FUNCTION_BLOCK FlushSludgeBuffer (* CAT Function Block Type *)
  (* Standard: 61499-2 *)
  (* Version 0.0, 6/19/2026, Schneider Electric, template *)
  PACKAGE SE.Nereda;
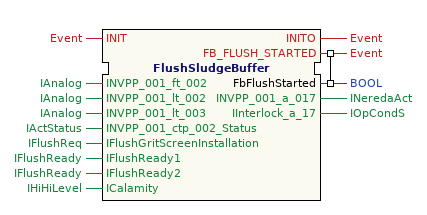
  EVENT_INPUT
    INIT;
  END_EVENT
  EVENT_OUTPUT
    INITO;
    FB_FLUSH_STARTED WITH FbFlushStarted;
  END_EVENT
  VAR_OUTPUT
    FbFlushStarted : BOOL;
  END_VAR
  SOCKETS
    INVPP_001_ft_002 : IAnalog;
    INVPP_001_lt_002 : IAnalog;
    INVPP_001_lt_003 : IAnalog;
    INVPP_001_ctp_002_Status : IActStatus;
    IFlushGritScreenInstallation : IFlushReq;
    IFlushReady1 : IFlushReady;
    IFlushReady2 : IFlushReady;
    ICalamity : IHiHiLevel;
  END_SOCKETS
  PLUGS
    INVPP_001_a_017 : INeredaAct;
  END_PLUGS
  PLUGS
    IInterlock_a_17 : IOpCondS; (* Condition summary chain output to downstream block *)
  END_PLUGS
  (* 01 - FUNCTIONNAL INPUT INTERFACE *)
  (* 00 - INITIALIZATION *)
  (* 05 - LOGIC *)
  (* 06 - HMI INTERFACE *)
  (* 03 - FIELD INTERFACE *)
  (* Grit Screens Flush Conditions *)
  (* 02 - FUNCTIONNAL OUTPUT INTERFACE *)
  (* Grit Screens Flush Control *)
  (* Interlock *)
  FBS
    FlushConditions : FlushCdt(pin_AD4F1D04748929A2 := 'Effluent Level is ok', pin_D80C7C0ABBECCDAB := 'Sludge Buffer Flushing', pin_E55C299A5BCFE2A5 := 'NVPP 001 a-- 017 is Available', pin_4F5AA965534A9167 := 'No Low Low Flow Alarm (Effluent Pump)', pin_D8438E8592CCBB68 := 'Effluent Pump is Ready', pin_F9CA602A9987631B := 'Flushing Parametrization is Done', pin_D946781DFBE190E0 := 'No Hi Level - Sludge Buffer', pin_2F47EB70426E0A5E := 'Flush Level Sp reached', pin_2D24E9AB41BE5BDB := TRUE, pin_EDFD852BF7F500FC := '');
    IThis : FlushSludgeBuffer_HMI(QI := TRUE);
    NVPP_001_lt_002_Status : decodeStatus; {SET_ATTRIBUTE(Configuration.Component.HideUnusedPorts, )}
    NotLowLevel : NOT_42C76073DCEB1A7A; {SET_ATTRIBUTE(Configuration.GenericFBType.InterfaceParams, Runtime.Standard#CNT:=1;OUT${CNT$}:BOOL)}
    GritScreensFlushControl : FlushingManagerSLB;
    Valve016_002Cmd : boolValueChanged;
    DurationSp : COMPARE_231D1C451B8C01CD0(IN2 := T#0ms); {SET_ATTRIBUTE(Configuration.GenericFBType.InterfaceParams, Runtime.Standard#CNT:=2;IN${CNT$}:TIME)} {SET_ATTRIBUTE(Configuration.Component.HideUnusedPorts, )}
    ConfigDone : AND_88A3DD8EC65DD11C; {SET_ATTRIBUTE(Configuration.GenericFBType.InterfaceParams, Runtime.Standard#CNT:=2;OUT:BOOL)}
    NVPP_001_ft_002_Status : decodeStatus; {SET_ATTRIBUTE(Configuration.Component.HideUnusedPorts, )}
    NotLowLowFlow : NOT_42C76073DCEB1A7A; {SET_ATTRIBUTE(Configuration.GenericFBType.InterfaceParams, Runtime.Standard#CNT:=1;OUT${CNT$}:BOOL)}
    CmdValve016_002 : BOOL2INT;
    FlowSp : COMPARE_1329C2AB45109BAAB(IN2 := 0); {SET_ATTRIBUTE(Configuration.GenericFBType.InterfaceParams, Runtime.Standard#CNT:=2;IN${CNT$}:REAL)} {SET_ATTRIBUTE(Configuration.Component.HideUnusedPorts, )}
    ForceStopSmooth : boolValueChanged;
    ForceStop : OR_NOT(pin_5391A9290C426EAD := FALSE, pin_0C6244A1FA53F771 := FALSE, pin_C718A4E0F6B1A5AF := FALSE, pin_F9B6B2F79CE46D8A := FALSE, pin_892061249439E371 := FALSE, pin_A17BF02B1ECA9592 := FALSE, pin_8BCAE36E149A36F2 := FALSE, pin_58FCE90E3A313BCD := TRUE, pin_7433DE8044744DCF := FALSE, pin_8555750E45CD1B5C := TRUE);
    ResetBtns : RESET_BTNs;
    NVPP_001_lt_003_Status : decodeStatus; {SET_ATTRIBUTE(Configuration.Component.HideUnusedPorts, )}
    NoHiLevel : NOT_42C76073DCEB1A7A; {SET_ATTRIBUTE(Configuration.GenericFBType.InterfaceParams, Runtime.Standard#CNT:=1;OUT${CNT$}:BOOL)}
    FlushStartLevelSp : COMPARE_1329C2AB45109BAAB; {SET_ATTRIBUTE(Configuration.GenericFBType.InterfaceParams, Runtime.Standard#CNT:=2;IN${CNT$}:REAL)}
    HighHighLevel_Calamity : ilckCondItem(CondCause := Active1);
    HighHighCalamity : OR_88A3DD8EC65DD11C; {SET_ATTRIBUTE(Configuration.GenericFBType.InterfaceParams, Runtime.Standard#CNT:=2;OUT:BOOL)}
    Wait : E_DELAY(DT := T#10s);
    GSsORGSsStarted : OR_88A3DD8EC65DD11C; {SET_ATTRIBUTE(Configuration.GenericFBType.InterfaceParams, Runtime.Standard#CNT:=2;OUT:BOOL)}
    DurationTime : E_DELAY_HOLD_V_D;
    Smooth : boolValueChanged;
    GSsORGSsFlushStarted : OR_88A3DD8EC65DD11C; {SET_ATTRIBUTE(Configuration.GenericFBType.InterfaceParams, Runtime.Standard#CNT:=2;OUT:BOOL)}
    Smooth1 : boolValueChanged;
  END_FBS
  EVENT_CONNECTIONS
    INVPP_001_lt_002.REQ_STATUS TO NVPP_001_lt_002_Status.REQ;
    NVPP_001_lt_002_Status.CNF TO NotLowLevel.REQ;
    NotLowLowFlow.CNF TO DurationSp.REQ;
    DurationSp.CNF TO FlowSp.REQ;
    INVPP_001_ft_002.REQ_STATUS TO NVPP_001_ft_002_Status.REQ;
    NVPP_001_ft_002_Status.CNF TO NotLowLevel.REQ;
    NotLowLevel.CNF TO NotLowLowFlow.REQ;
    FlushConditions.E74FDFC5C9E17061 TO INITO;
    DurationTime.INITO TO FlushConditions.7689825C23C7E3C1;
    INVPP_001_a_017.9CD053F8408797ED TO GritScreensFlushControl.17EF565317C21577;
    DurationTime.1457E63E0C241C83 TO GritScreensFlushControl.6BFDB43937C58B53;
    GritScreensFlushControl.FB17218C6899B6C2 TO FB_FLUSH_STARTED;
    GritScreensFlushControl.7C8478AB3E0AC40C TO Valve016_002Cmd.REQ;
    GritScreensFlushControl.4439D0346679ABD7 TO IFlushGritScreenInstallation.058C8BB5EF4C4954;
    GritScreensFlushControl.CNF_FLUSH_START TO DurationTime.START;
    GritScreensFlushControl.CNF_FLUSH_STOP TO DurationTime.STOP;
    Valve016_002Cmd.CHD TO CmdValve016_002.DD5870AA881150BB;
    CmdValve016_002.6FC99A5BD1C38561 TO INVPP_001_a_017.0F1CDF9A9B4A227A;
    INVPP_001_a_017.CC753684FA882790 TO NotLowLevel.REQ;
    FlushStartLevelSp.CNF TO FlushConditions.C4A26A2931936C6C;
    ForceStop.5E2BC6C1897CC372 TO ForceStopSmooth.REQ;
    FlushConditions.144BD964598CDC30 TO GritScreensFlushControl.D472A6751679CB56;
    INIT TO IThis.1EF99DCB15A49BE4;
    GritScreensFlushControl.GRAPH TO IThis.623B20E659F013A2;
    FlushConditions.E74FDFC5C9E17061 TO IThis.6CA585F7EA2251CC;
    ResetBtns.920962203CA54948 TO IThis.BC4D95AF9C39047B;
    IThis.97A2502A32C860AE TO DurationTime.INIT;
    IThis.40B0BCBFC46CBB6D TO NotLowLevel.REQ;
    IThis.40B0BCBFC46CBB6D TO IFlushGritScreenInstallation.A591EFC748C65FB0;
    IThis.40B0BCBFC46CBB6D TO DurationTime.8C325F07198FCB13;
    IThis.C0957A1C40CEA3B4 TO GritScreensFlushControl.F40A51463574875E;
    IThis.C0957A1C40CEA3B4 TO ResetBtns.AB695E9A35A20E19;
    GritScreensFlushControl.F622B0785D87399D TO IFlushGritScreenInstallation.91C62E5F9EC3AD97;
    INVPP_001_ctp_002_Status.14377629A1F197A9 TO NotLowLevel.REQ;
    IFlushGritScreenInstallation.158ACCEF11EA11F4 TO GritScreensFlushControl.2E9E428AF53DA484;
    INVPP_001_lt_003.REQ_STATUS TO NVPP_001_lt_003_Status.REQ;
    NVPP_001_lt_003_Status.CNF TO NotLowLevel.REQ;
    ForceStopSmooth.CNF TO NoHiLevel.REQ;
    NoHiLevel.CNF TO FlushStartLevelSp.REQ;
    INVPP_001_lt_003.REQ TO NotLowLevel.REQ;
    FlushStartLevelSp.CNF TO GritScreensFlushControl.7CCDF8BA66CD247C;
    HighHighCalamity.CNF TO HighHighLevel_Calamity.REQ;
    ICalamity.15126F43E529BB4F TO HighHighCalamity.REQ;
    FlowSp.CNF TO ConfigDone.REQ;
    ConfigDone.CNF TO ForceStop.AE1B4DCC5DF54611;
    GritScreensFlushControl.9781ED32849F99B4 TO Wait.START;
    Wait.EO TO GritScreensFlushControl.F24FFDC5DA37517C;
    IFlushReady1.EB400628E9D6A506 TO GSsORGSsStarted.REQ;
    IFlushReady2.EB400628E9D6A506 TO GSsORGSsStarted.REQ;
    GritScreensFlushControl.33239982CC8E7419 TO DurationTime.46FF7A1A69D9FEE0;
    GSsORGSsStarted.CNF TO Smooth.REQ;
    Smooth.CHD TO GritScreensFlushControl.D472A6751679CB56;
    IFlushReady1.A6EF038FCF65FFCE TO GSsORGSsFlushStarted.REQ;
    IFlushReady2.A6EF038FCF65FFCE TO GSsORGSsFlushStarted.REQ;
    GSsORGSsFlushStarted.CNF TO Smooth1.REQ;
    Smooth1.CHD TO GritScreensFlushControl.C7A0D51879FE2FD9;
  END_CONNECTIONS
  DATA_CONNECTIONS
    INVPP_001_lt_002.Status TO NVPP_001_lt_002_Status.Status;
    NVPP_001_lt_002_Status.LoAlarm TO NotLowLevel.IN1;
    INVPP_001_ft_002.Status TO NVPP_001_ft_002_Status.Status;
    NVPP_001_ft_002_Status.LoLoAlarm TO NotLowLowFlow.IN1;
    NotLowLevel.OUT1 TO FlushConditions.22A84A30EE8DD605;
    INVPP_001_a_017.8A8A07EFCDA1443C TO FlushConditions.4ED40FD24D2392DA;
    NotLowLowFlow.OUT1 TO FlushConditions.504E64E2CDCF5D86;
    INVPP_001_ctp_002_Status.9E0B44559326BEAF TO FlushConditions.9BB2492C130556E4;
    GritScreensFlushControl.7925856953128FBE TO FbFlushStarted;
    GritScreensFlushControl.6EFD4A5711C4475D TO Valve016_002Cmd.Input;
    GritScreensFlushControl.D35FF54DD8CD3DCD TO IFlushGritScreenInstallation.78ED129B4768A8A1;
    GritScreensFlushControl.809D6A4978DE08CF TO IFlushGritScreenInstallation.23612E77D592C190;
    Valve016_002Cmd.Output TO CmdValve016_002.4573FC8F228EB71D;
    DurationTime.716D3F3042596C89 TO GritScreensFlushControl.FlushDurationDone;
    INVPP_001_a_017.7F6CC7FEB9223DF3 TO GritScreensFlushControl.B4CCB3C919A81AAD;
    INVPP_001_a_017.A8D6C4A1FDCCA991 TO GritScreensFlushControl.927265D5AE017F25;
    IFlushGritScreenInstallation.309BBEDA7DF51DE0 TO GritScreensFlushControl.EB78D4EC51374885;
    IFlushGritScreenInstallation.E3447F193E0C5923 TO GritScreensFlushControl.8C9A5C84A4BBC11A;
    IFlushGritScreenInstallation.102FEFFE81A835E5 TO GritScreensFlushControl.BE830E3A77806910;
    IFlushGritScreenInstallation.32E78DF7D9CBD985 TO GritScreensFlushControl.CA6B1E62BFF3D73B;
    CmdValve016_002.A6DEF5F9C27C1848 TO INVPP_001_a_017.710D7FC54EE3F35A;
    ForceStop.39A6EB2EA34CB8B9 TO ForceStopSmooth.Input;
    NotLowLevel.OUT1 TO ForceStop.305F82B0106D312B;
    INVPP_001_a_017.8A8A07EFCDA1443C TO ForceStop.DD1680AE8DA8DF87;
    NotLowLowFlow.OUT1 TO ForceStop.92ECDEDDB24CC262;
    INVPP_001_ctp_002_Status.9E0B44559326BEAF TO ForceStop.2CF1E7F52666F162;
    FlushConditions.5C1922DA22925005 TO GritScreensFlushControl.EnableOperation;
    GritScreensFlushControl.Grafcet TO IThis.4EF02231C06E8D13;
    IThis.1AA6078AD289AF22 TO DurationSp.IN1;
    IThis.1AA6078AD289AF22 TO DurationTime.DT1;
    IThis.3E1384426DD858B0 TO FlowSp.IN1;
    IThis.3E1384426DD858B0 TO IFlushGritScreenInstallation.34B76CCA964D89EE;
    IThis.CEC3C53B3ACE8E6D TO GritScreensFlushControl.0FA765E9822F7BA9;
    IThis.CEC3C53B3ACE8E6D TO ResetBtns.479D4538AEFD6EE1;
    IThis.1BFB680DD0A7C843 TO GritScreensFlushControl.3C22F17908DBA162;
    GritScreensFlushControl.51D0A2C29DC62FA2 TO IFlushGritScreenInstallation.B5CD30493D22784A;
    GritScreensFlushControl.7AB11AE4573B259E TO IFlushGritScreenInstallation.10050E1891596878;
    IFlushGritScreenInstallation.0154EF4D281C90FC TO GritScreensFlushControl.9CD632B5AC2CF415;
    INVPP_001_lt_003.Status TO NVPP_001_lt_003_Status.Status;
    NVPP_001_lt_003_Status.HiAlarm TO NoHiLevel.IN1;
    NoHiLevel.OUT1 TO FlushConditions.4E3CFAB7818DC81F;
    FlushStartLevelSp.LE TO FlushConditions.47969CBC2D520AAD;
    INVPP_001_lt_003.Value TO FlushStartLevelSp.IN1;
    IThis.34A2F2095903B30B TO FlushStartLevelSp.IN2;
    FlushStartLevelSp.GT TO GritScreensFlushControl.336396CDA8290477;
    FlushStartLevelSp.LE TO GritScreensFlushControl.B610A3A56F10FBA2;
    HighHighCalamity.OUT TO HighHighLevel_Calamity.CondSignal;
    ICalamity.C818324478A2F205 TO HighHighCalamity.IN1;
    ICalamity.96B50ADF37756FFC TO HighHighCalamity.IN2;
    DurationSp.NE TO ConfigDone.IN1;
    FlowSp.NE TO ConfigDone.IN2;
    ConfigDone.OUT TO FlushConditions.9D55FD7AD1246DA2;
    ConfigDone.OUT TO ForceStop.4997B302A4472F6A;
    IFlushGritScreenInstallation.F75B2D6279DB7772 TO GritScreensFlushControl.AED40E274B455BA3;
    IFlushGritScreenInstallation.FBD19C5680BE3A13 TO GritScreensFlushControl.266B23EDF02E98D5;
    IFlushReady1.948E4422D799D3D4 TO GSsORGSsStarted.IN1;
    IFlushReady2.948E4422D799D3D4 TO GSsORGSsStarted.IN2;
    Smooth.Output TO GritScreensFlushControl.6757599E742CC6CD;
    GritScreensFlushControl.FDBF246FF450FFC3 TO DurationTime.5F12F87EEE9002AF;
    GSsORGSsStarted.OUT TO Smooth.Input;
    IFlushReady1.3B406C848FF944CA TO GSsORGSsFlushStarted.IN1;
    IFlushReady2.3B406C848FF944CA TO GSsORGSsFlushStarted.IN2;
    GSsORGSsFlushStarted.OUT TO Smooth1.Input;
    Smooth1.Output TO GritScreensFlushControl.1290DB47BB4481FA;
  END_CONNECTIONS
  ADAPTER_CONNECTIONS
    HighHighLevel_Calamity.ICondChainOut TO IInterlock_a_17;
  END_CONNECTIONS
END_FUNCTION_BLOCK
